TYPE HydraulicsStatuses :
STRUCT
	initializationStatus: InitializationStatus;
	healthStatus: HealthStatus;
	busyStatus: BusyStatus;
	operatingStatus: OperatingStatus;
END_STRUCT
END_TYPE

(* stored: Version 1.1.0.1, ProductVersion 3.1.4019.2
   DUT HydraulicsStatuses: Id {fd4d5cde-36bf-40ae-be2c-adf6bdff9c04} *)
